TYPE AbsPosition :
STRUCT
	x:LREAL;
	y:LREAL;
	z:LREAL;
END_STRUCT
END_TYPE

(* stored: Version 1.1.0.1, ProductVersion 3.1.4022.12
   DUT AbsPosition: Id {80d954a6-a2b2-414e-b152-0dbb418b306e} *)
